SYSTEM ConnectionRepairTest
  (* Version 1.0, 2026-07-21, Dimitrios Kalligaridis *)
  APPLICATION App
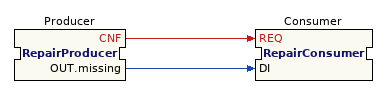
    FBS
      Producer : RepairProducer;
      Consumer : RepairConsumer;
    END_FBS
    EVENT_CONNECTIONS
      Producer.CNF TO Consumer.REQ;
    END_CONNECTIONS
    DATA_CONNECTIONS
      Producer.OUT.missing TO Consumer.DI;
    END_CONNECTIONS
  END_APPLICATION
END_SYSTEM
